// TIA Portal V17 export
// export: Created 2025-03-05T08:00:48.1691025Z, ExportSetting WithDefaults, DisplayName Totally Integrated Automation Portal, DisplayVersion V17 Update 8, DisplayName TIA Portal Openness, DisplayVersion V17 Update 8, DisplayName TIA Portal Version Control Interface, DisplayVersion V17, DisplayName SINAMICS Startdrive Advanced, DisplayVersion V17 SP2, DisplayName SINAMICS Startdrive G110M, G120, G120C, G120D, G120P, G115D, DisplayVersion V17 SP2, DisplayName SINAMICS Startdrive G130, G150, S120, S150, SINAMICS MV, S210, DisplayVersion V17 SP2, DisplayName STEP 7 Professional, DisplayVersion V17 Update 8, DisplayName SINUMERIK ONE STEP 7 Toolbox, DisplayVersion V17 Update 12, DisplayName SINUMERIK 840D sl STEP 7 Toolbox, DisplayVersion V17 Update 12, DisplayName STEP 7 Safety, DisplayVersion V17 Update 6, DisplayName WinCC Advanced, DisplayVersion V17 Update 8
DATA_BLOCK "DB1401_PNEUMATIC_SYSTEM"   // DB1401
{ DB_Accessible_From_OPC_UA := 'FALSE' }
AUTHOR : ETXETAR
VERSION : 1.0
// stored: AutoNumber false, DBAccessibleFromOPCUA false, DBAccessibleFromWebserver true, InstanceOfName FB1401_PNEUMATIC_SYSTEM, InstanceOfType FB
"FB1401_PNEUMATIC_SYSTEM"
   // VAR_INPUT
   //    OPTIONS_0 : Byte;
   //    OPTIONS_1 : Byte;
   //    OPTIONS_2 : Byte;
   //    PRESSURE : Bool;
   //    DRIVE_UNBLOCKED : Bool;
   //    CONNECTION_1_SENSOR : Bool;
   //    CONNECTION_2_SENSOR : Bool;
   //    FLOW_SENSOR : UInt;
   //    TEMPERATURE_SENSOR : UInt;
   //    PRESSURIZED : Bool;
   //    U01_GRIPPER_PRESSURIZED : Bool;
   //    U01_LABERINT_PRESSURIZED : Bool;
   //    U01_UPPER_TABLE_PRESSURIZED : Bool;
   //    U01_LOWER_TABLE_PRESSURIZED : Bool;
   //    U01_CART_X_PRESSURIZED : Bool;
   //    U01_STA_3_MEAS_PRESSURIZED : Bool;
   //    U02_GRIPPER_PRESSURIZED : Bool;
   //    U02_LABERINT_PRESSURIZED : Bool;
   //    U02_UPPER_TABLE_PRESSURIZED : Bool;
   //    U02_LOWER_TABLE_PRESSURIZED : Bool;
   //    U02_CART_X_PRESSURIZED : Bool;
   //    U02_STA_3_MEAS_PRESSURIZED : Bool;
   //    HMI_REQ_LINE : Bool;
   // END_VAR
   // VAR_OUTPUT
   //    HMI_POWER_UP_COND_OFF : Bool;
   //    HMI_POWER_UP_COND_ON : Bool;
   //    HMI_POWER_UP_EXECU_LEFT : Bool;
   //    HMI_POWER_UP_EXECU_RIGHT : Bool;
   //    MAIN_VALVE : Bool;
   //    CONNECTION_1 : Bool;
   //    CONNECTION_2 : Bool;
   //    PRESSURIZATION_ON : Bool;
   //    PRESSURIZATION_OFF : Bool;
   //    DRIVE_UNBLOCK : Bool;
   // END_VAR
   // VAR RETAIN
   //    AIR_FLOW_VALUE : Real;
   //    TEMPERATURE_VALUE : Real;
   //    PRESS_NOT_REACHED_ALARM : Bool;
   //    PRESS_SWITCH_ALARM : Bool;
   //    PRESS_MISSING_ALARM : Bool;
   //    CONNECTION_SENSOR_1_ALARM : Bool;
   //    CONNECTION_SENSOR_2_ALARM : Bool;
   //    UNBLOCK_DRIVE_PRESS_ALARM : Bool;
   //    UNBLOCK_DRIVE_PRESS_SWITCH_ALARM : Bool;
   //    PRESSURIZATION_ALARM : Bool;
   //    PRESSURIZATION_SWITCH_ALARM : Bool;
   //    PNEUMATIC_TEMPERATURE_INPUT_ALARM : Bool;
   //    PNEUMATIC_FLOW_INPUT_ALARM : Bool;
   //    U01_GRIPPER_PRESSURIZATION_ALARM : Bool;
   //    U01_GRIPPER_PRESSURIZATION_SWITCH_ALARM : Bool;
   //    U01_LABERINT_PRESSURIZATION_ALARM : Bool;
   //    U01_LABERINT_PRESSURIZATION_SWITCH_ALARM : Bool;
   //    U01_UPPER_TABLE_PRESSURIZATION_ALARM : Bool;
   //    U01_UPPER_TABLE_PRESSURIZATION_SWITCH_ALARM : Bool;
   //    U01_LOWER_TABLE_PRESSURIZATION_ALARM : Bool;
   //    U01_LOWER_TABLE_PRESSURIZATION_SWITCH_ALARM : Bool;
   //    U01_CART_AXIS_X_PRESSURIZATION_ALARM : Bool;
   //    U01_CART_AXIS_X_PRESSURIZATION_SWITCH_ALARM : Bool;
   //    U01_STA_3_MEAS_PRESSURIZATION_ALARM : Bool;
   //    U01_STA_3_MEAS_PRESSURIZATION_SWITCH_ALARM : Bool;
   //    U02_GRIPPER_PRESSURIZATION_ALARM : Bool;
   //    U02_GRIPPER_PRESSURIZATION_SWITCH_ALARM : Bool;
   //    U02_LABERINT_PRESSURIZATION_ALARM : Bool;
   //    U02_LABERINT_PRESSURIZATION_SWITCH_ALARM : Bool;
   //    U02_UPPER_TABLE_PRESSURIZATION_ALARM : Bool;
   //    U02_UPPER_TABLE_PRESSURIZATION_SWITCH_ALARM : Bool;
   //    U02_LOWER_TABLE_PRESSURIZATION_ALARM : Bool;
   //    U02_LOWER_TABLE_PRESSURIZATION_SWITCH_ALARM : Bool;
   //    U02_CART_AXIS_X_PRESSURIZATION_ALARM : Bool;
   //    U02_CART_AXIS_X_PRESSURIZATION_SWITCH_ALARM : Bool;
   //    U02_STA_3_MEAS_PRESSURIZATION_ALARM : Bool;
   //    U02_STA_3_MEAS_PRESSURIZATION_SWITCH_ALARM : Bool;
   //    SWITCH_ON_GENERAL_CONDITIONS : Bool;
   //    SWITCH_ON_INITIAL_CONDITIONS : Bool;
   //    SWITCH_ON_MANUAL_REQUEST : Bool;
   //    SWITCH_ON_AUTO_REQUEST : Bool;
   //    SWITCH_ON_GLOBAL_REQUEST : Bool;
   //    SWITCH_ON_COMMAND : Bool;
   //    SWITCH_ON : Bool;
   //    IN_SERVICE : Bool;
   //    SWITCH_OFF_GENERAL_CONDITIONS : Bool;
   //    SWITCH_OFF_INITIAL_CONDITIONS : Bool;
   //    SWITCH_OFF_MANUAL_REQUEST : Bool;
   //    SWITCH_OFF_AUTO_REQUEST : Bool;
   //    SWITCH_OFF_GLOBAL_REQUEST : Bool;
   //    SWITCH_OFF_COMMAND : Bool;
   //    SWITCH_OFF : Bool;
   //    OUT_OF_SERVICE : Bool;
   //    MANUAL_REQUEST_HELP : Bool;
   //    SWITCH_ON_GENERAL_CONDITION_HELP : Bool;
   //    SWITCH_ON_INITIAL_CONDITION_HELP : Bool;
   //    SWITCH_OFF_GENERAL_CONDITION_HELP : Bool;
   //    SWITCH_OFF_INITIAL_CONDITION_HELP : Bool;
   //    ANY_ACTIVE_ALARM : Bool;
   //    IS_ALARMS : Bool;
   //    SEOC_ALARMS : Bool;
   //    WARNINGS : Bool;
   //    WARNINGS_GONE : Bool;
   //    TIMER_PRESSURE_ALARM : TON_TIME;
   //    TIMER_PRESSURE_SWITCH_ALARM : TON_TIME;
   //    TIMER_PRESSURE_MISSING_ALARM : TON_TIME;
   //    TIMER_CONNECTION_SENSOR_1_ALARM : TON_TIME;
   //    TIMER_CONNECTION_SENSOR_1_SWITCH_ALARM : TON_TIME;
   //    TIMER_CONNECTION_SENSOR_2_ALARM : TON_TIME;
   //    TIMER_CONNECTION_SENSOR_2_SWITCH_ALARM : TON_TIME;
   //    TIMER_DRIVE_PRESSURE_UNBLOCK_ALARM : TON_TIME;
   //    TIMER_DRIVE_PRESSURE_UNBLOCK_SWITCH_ALARM : TON_TIME;
   //    TIMER_PRESSURE_ON_DEVICES : TON_TIME;
   //    TIMER_PRESSURE_OFF_DEVICES : TON_TIME;
   //    TIMER_PRESSURIZATION_OFF_DELAY { S7_SetPoint := 'True'} : TOF_TIME;
   // END_VAR
BEGIN
END_DATA_BLOCK
